FUNCTION_BLOCK kalmanController
VAR_INPUT
END_VAR
VAR_OUTPUT
END_VAR
VAR
	 linSpdCommand,fwdMoveSpdCommand,angMoveSpdCommand,angFwdPosError,angMovePosError,angFwdPosCommand,linSpdCommandShaped,linMoveSpdCommand,angSpdCommand:LREAL;
	 missionCompletedAng,missionCompletedLin:INT;
	 fb_kinematicSolution:kinematicSolution;
	 fb_localization:localization;
	 FB_DRIVE_MOTORS:DriveMotors();
END_VAR

IF (robotdata.motion_status = MOTION_ONGOING OR robotdata.motion_status = MOTION_ANGLE) AND (robotdata.activecommand=COMMAND_X_CORR OR robotdata.activecommand=COMMAND_ANG_CORR) THEN
	FB_DRIVE_MOTORS();


ELSIF(robotdata.controller=1)THEN
    fb_localization();
    missionCompletedLin := linPosErrGenerator(idealAngle,xGoal,yGoal,PosFdbckX,PosFdbckY,modeEnable);
    linMoveSpdCommand:= linPosErr* LINPOS_Kp;
    linSpdCommand := linSpdCommandMixer(modeEnable,linMoveSpdCommand,linPosErr);
    linSpdCommandShaped := linSpdCommandLimiter(linSpdCommand);
    angFwdPosCommand := forwardMovement(PosFdbckX,PosFdbckY,idealAngle);
    angMovePosError := angErrorCalc(AngPosCommand,robotAngle);
    angFwdPosError := angErrorCalc(angFwdPosCommand,robotAngle);
    angMoveSpdCommand := angMovePosError * TURNANG_Kp;
    fwdMoveSpdCommand := angFwdPosError* TURNFWD_Kp;
    
    missionCompletedAng:=angSpdCommandMixer(angMovePosError,modeEnable,angMoveSpdCommand,fwdMoveSpdCommand,angSpdCommand);
    angSpdCommandLimiter(angSpdCommand);
    missionCompleted:=(missionCompletedAng OR missionCompletedLin);
    IF(missionCompleted=1) THEN
		robotdata.motion_status:=MOTION_ENDED;
	END_IF
 
    fb_kinematicSolution(linSpdCommandShaped:=linSpdCommandShaped,angSpdCommand:=angSpdCommandShaped);

    IF (missionCompleted=1) THEN
       
      robotdata.motion_status := MOTION_ENDED;
	  robotdata.activeState:=MOVE_ENDED;
	  robotdata.Position_Velocity.Locomotion_1_target_velocity:= 0;
	  robotdata.Position_Velocity.Locomotion_2_target_velocity:= 0;
	  ELSE
		robotdata.Position_Velocity.Locomotion_1_target_velocity := leftMotorSpeedCommand;
		robotdata.Position_Velocity.Locomotion_2_target_velocity:=-1*rightMotorSpeedCommand;
	 END_IF
  END_IF

END_FUNCTION_BLOCK

(* stored: Version 1.1.0.1, ProductVersion 3.1.4024.12
   POU kalmanController: Id {d981cfdb-89fe-46a7-b0aa-9698b864aae4}, SpecialFunc None *)
